{attribute 'pack_mode' := '1'}
TYPE stEL9576 :
STRUCT
    BCT_Inputs AT %I* : stEL9576_Status;
END_STRUCT
END_TYPE;

(* stored: Version 1.1.0.1, ProductVersion 3.1.4024.4
   DUT stEL9576: Id {3f662b74-2f63-4648-9b5f-3f1e403de529} *)
